{attribute 'qualified_only'}
{attribute 'to_string'}
TYPE E_JointStates :
(
	Idle:=0,
	Setup1,
	Setup2
)UINT := Idle
;
END_TYPE

(* stored: Version 1.1.0.1, ProductVersion 3.1.4024.12
   EnumerationTextList E_JointStates: Id {7fc3575a-2c52-4b3c-bd8b-0056d68a78d6} *)
